Yaskawa INFORM job: AAA.JBI

/JOB
//NAME AAA
//POS
///NPOS 2,0,0,0,0,0
C00000=-29502,67644,32784,10511,-54069,-12462
C00001=0,0,0,0,0,0
//INST
///DATE 2023/03/21 13:13
///ATTR SC,RW
///GROUP1 RB1
NOP
'Using Motoman MA2010 Base (ta
'rgets wrt base):
'0.0,0.0,0.0,0.0,0.0,0.0
MOVJ C00000 VJ=10.0
MOVJ C00001 VJ=8.0
END
